// SIMATIC S7-200 project (STEP 7-Micro/WIN), CPU 224 REL 02.00

ORGANIZATION_BLOCK MAIN:OB1
TITLE=这是一个化工厂中的液体混合装置，用于将两种化学液体按一定比例混合，应用于生产特定化学产品的场景。此外，由于化学反应需要控制温度在200°C至220°C的适宜范围内进行，我们额外增加加热器和冷却器以控制反应温度，避免不必要的能源浪费。设计程序依赖温度传感器调整加热器和冷却器的单独开关，以防加热器和冷却器的同步启动。
// 
// 系统通过启动按钮启动混合过程，首先打开进料阀门A控制和进料阀门B控制进行进料，直至液位传感器检测到液位达到预设值。
// 进料启用标志只有在液位传感器未检测到满液位且液位未满标志未置位时才能置位，防止混合罐溢出。
// 进料过程中，系统监控温度，确保混合在200°C至220°C的适宜范围内进行。
// 若温度低于200°C，激活加热器；若温度高于220°C，激活冷却系统。
// 进料阀门A,B置位的前提都需要保证在温度适宜的情况下。
// 进料阀门A控制在启动脉冲为真触发；并且受进料A控制和进料延时定时器影响持续保持置位状态。
// 进料阀门B控制由模式切换脉冲为真时触发；
// 进料完成后，系统启动搅拌电机控制进行搅拌，搅拌时间由搅拌延时定时器控制60个时间单位。
// 搅拌电机控制只能在搅拌启用标志置位且温度适宜时激活，并在进料延时定时器到时或停止脉冲置位时复位，保证搅拌过程在规定时间和温度条件下完成。
// 搅拌结束后，打开出料阀门控制进行出料，出料阀门控制必须在复位脉冲置位时打开，并在搅拌延时定时器到时或停止脉冲置位时关闭，确保混合液体在搅拌完成后安全输出。
// 停止按钮可随时停止整个过程，复位按钮将系统复位到初始状态，手动/自动切换开关允许操作员选择手动或自动模式。
BEGIN
Network 1
LD     I0.0
EU
=      M10.0
?000
Network 2
LD     I0.1
EU
=      M10.1
Network 3
LD     I0.2
EU
=      M10.2
Network 4
LD     I0.3
EU
=      M10.3
Network 5
LDN    I0.4
AN     M11.3
=      M11.2
Network 6
LDN    I0.4
=      M11.3
Network 7
LD     M10.0
S      M20.0, 1
Network 8
LD     M20.0
A      T38
O      M10.0
A      M30.0
S      Q0.0, 1
Network 9
LD     M10.3
A      M30.0
S      Q0.1, 1
Network 10
LD     M10.3
O      M10.1
R      Q0.0, 1
Network 11
LD     M10.2
S      Q0.3, 1
Network 12
LD     M11.4
A      M30.0
S      Q0.4, 1
Network 13
LD     M10.2
O      M10.1
R      Q0.1, 1
Network 14
LD     T37
O      M10.1
R      Q0.3, 1
Network 15
LD     Q0.3
TON    T37, +60
Network 16
LDN    Q0.3
=      M12.4
Network 17
LDN    Q0.3
A      M12.4
AN     M11.5
=      M11.4
Network 18
LDN    Q0.3
A      M12.4
=      M11.5
Network 19
LD     M11.4
A      M30.0
S      Q0.2, 1
Network 20
LD     T38
O      M10.1
R      Q0.2, 1
Network 21
LD     M11.2
S      M20.1, 1
Network 22
LD     T38
R      M20.1, 1
Network 23
LD     M20.1
TON    T38, +20
Network 24
LDB<   VB800, 200
=      Q1.1
Network 25
LDB>   VB800, 220
=      Q1.2
Network 26
LDN    Q1.1
AN     Q1.2
=      M30.0
END_ORGANIZATION_BLOCK
